FUNCTION_BLOCK FB_Gate
VAR_INPUT
	GateStat:BOOL;
	GatePosition:INT;
	GateTimer:TON;
END_VAR

END_FUNCTION_BLOCK

(* stored: Version 1.1.0.1, ProductVersion 3.1.4024.3
   POU FB_Gate: Id {5dd372f6-e7bc-4901-9720-6b285220b02e}, SpecialFunc None *)
